FUNCTION_BLOCK AddMoverToGroupTask IMPLEMENTS ITask
VAR_INPUT
END_VAR
VAR_OUTPUT
END_VAR
VAR
	AddtoGrp			: MC_AddAxisToGroup;
	_caGroup			: ICollisionGroup;
	_axis				: reference TO AXIS_REF;
	State: INT;
	_addMover : BOOL;
	_busy : BOOL;
	_error : BOOL;
	_done : BOOL;
	_moverNumber : UDINT;
END_VAR

CASE State OF
	0:
		IF _addMover THEN
			_done := FALSE;
			_error := FALSE;
			_busy := true;
			AddtoGrp.Execute := TRUE;
			IF AddtoGrp.Busy THEN
				State := 10;
				_addMover := FALSE;
			END_IF
		END_IF
	
	10:
		IF NOT AddtoGrp.Busy THEN
			IF AddtoGrp.Done THEN
				_done := TRUE;
			ELSIF AddtoGrp.Error THEN
				_error := TRUE;
			END_IF
			_busy := FALSE;
			AddtoGrp.Execute := false;
			State := 0;
		END_IF
END_CASE

AddtoGrp(AxesGroup := _caGroup.GroupRef,
			Axis := _axis,
			IdentInGroup := UDINT_TO_IDENTINGROUP(_moverNumber));

METHOD Abort : BOOL
AddtoGrp.Execute := FALSE;
Abort := true;
State := 0;
END_METHOD

METHOD AddMover : BOOL
VAR_INPUT
	MoverToAdd : IMover;
END_VAR
_axis REF= MoverToAdd.AxisRef;
_moverNumber := INT_TO_UDINT(MoverToAdd.IdentInGroup);
_busy := TRUE;
AddMover := _addMover := TRUE;
END_METHOD

PROPERTY Busy : BOOL
GET
Busy := _busy;
END_GET
END_PROPERTY

PROPERTY Done : BOOL
GET
Done := _done;
END_GET
END_PROPERTY

PROPERTY Error : BOOL
GET
Error := _error;
END_GET
END_PROPERTY

METHOD FB_init : BOOL
VAR_INPUT
	bInitRetains : BOOL; // if TRUE, the retain variables are initialized (warm start / cold start)
	bInCopyCode : BOOL;  // if TRUE, the instance afterwards gets moved into the copy code (online change)
	collisionGroup : ICollisionGroup;	
END_VAR
_caGroup := collisionGroup;
END_METHOD

END_FUNCTION_BLOCK

(* stored: Version 1.1.0.1, ProductVersion 3.1.4024.11
   POU AddMoverToGroupTask: Id {feae89f9-a6fd-4234-9f55-63ef9d6596bc}, SpecialFunc None
   Method Abort: Id {ae830af7-f8b8-45b2-a2b9-e3017e78eb0f}
   Method AddMover: Id {51a205d2-594e-409d-8da4-1e5f87f7831a}
   Property Busy: Id {afcd1b54-e22b-49a3-9c9c-b3f0c79b4568}
   Get Get: Id {4b50b697-dd2d-42bd-9737-bd8b1caa6957}
   Property Done: Id {2659b571-fe6f-4583-a3e6-2e6986ef714f}
   Get Get: Id {2ae1ed02-cc28-4c24-8907-5b99691b0028}
   Property Error: Id {8e6f5a82-522c-424d-96f2-7406cd982aac}
   Get Get: Id {a14355d3-234a-4c04-9d54-25389bdf30c6}
   Method FB_init: Id {3a068e92-ba3f-4b22-90e4-bf7f0af1aaec} *)
